Yaskawa INFORM job: BABY.JBI

/JOB
//NAME BABY
//POS
///NPOS 7,0,0,0
///TOOL 0
///PULSE
C000=2331,39928,-20718,-4873,-947,6842
C001=795,48568,-54750,-12713,1069,8158
C002=-38334,51136,-52109,4254,4552,8821
C003=-38334,33280,-52109,4254,4552,8821
C004=-40062,38128,-17741,4898,7240,8765
C005=-13518,37984,-17597,5598,1444,8933
C006=-13518,37984,-54509,5598,1444,8933
//INST
///DATE 2014/09/13 22:59
///ATTR 0,0,0,0,0,0,0,0,0,0,0,0,0,1,0,0
///FRAME BASE
NOP
*F
MOVJ C000 VJ=50.00 CONT
MOVJ C001 VJ=50.00 CONT
MOVJ C002 VJ=100.00 CONT
MOVJ C003 VJ=100.00 CONT
MOVJ C004 VJ=100.00 CONT
MOVJ C005 VJ=50.00 CONT
MOVJ C006 VJ=50.00 CONT
JUMP *F
END
